{attribute 'qualified_only'}
VAR_GLOBAL
END_VAR

(* stored: Version 1.1.0.1, ProductVersion 3.1.4024.12
   GVL G_Input: Id {7bb65c8b-cba4-48b1-8daa-c9b33c78d82e} *)
